// TIA Portal V19 export
TYPE "LEXCHANGETRAY_typeConstraintWorkstation_deliver_interface"
// stored: Access Published
   STRUCT
      init : Bool;
      constraintRoller : "LEXCHANGETRAY_typeConstraintWorkstation_toConstraintRollerDeliver";
   END_STRUCT;
END_TYPE
